(* Logix 5000 project; controller Lab5 vendor 1 type 14 code 54 rev 16.20; software revision 16.03 *)

TASK MainTask (continuous, watchdog 500 ms) : MainProgram

MODULES
   Local : vendor 1 type 14 code 54 (ICP 0, rev 16.20)
       : vendor 1 type 7 code 2 (ICP 5, rev 3.1, Input RPI 20 ms)
       : 1756-OB16D (ICP 6, rev 3.1, Output RPI 20 ms)
END_MODULES

PROGRAM MainProgram   (* main routine MainRoutine *)
VAR
   Forward_Start_Pushbutton : ALIAS FOR Local:5:I.Data.0;
   M1_Forward_Motor_Starter : ALIAS FOR Local:6:O.Data.0;
   M2_Reverse_Motor_Starter : ALIAS FOR Local:6:O.Data.1;
   Motor_Running_Light : ALIAS FOR Local:6:O.Data.2;
   Motor_Stopped_Light : ALIAS FOR Local:6:O.Data.3;
   Reverse_Start_Pushbutton : ALIAS FOR Local:5:I.Data.1;
   srtbh : TIMER;
   Stop_Pushbutton : ALIAS FOR Local:5:I.Data.2;
   Time_Motor_Not_Running : TIMER;
   Time_Motor_Running : TIMER;
   Timer1 : TIMER := (PRE := 10000);
   Timer_Motor_Not_Running : TIMER := (PRE := 99999999, ACC := 3844);
   Timer_Motor_Running : TIMER := (PRE := 999999999);
   Toggle_Switch_1 : ALIAS FOR Local:5:I.Data.3;
   Toggle_Switch_2 : ALIAS FOR Local:5:I.Data.4;
END_VAR

ROUTINE MainRoutine   (* ladder *)
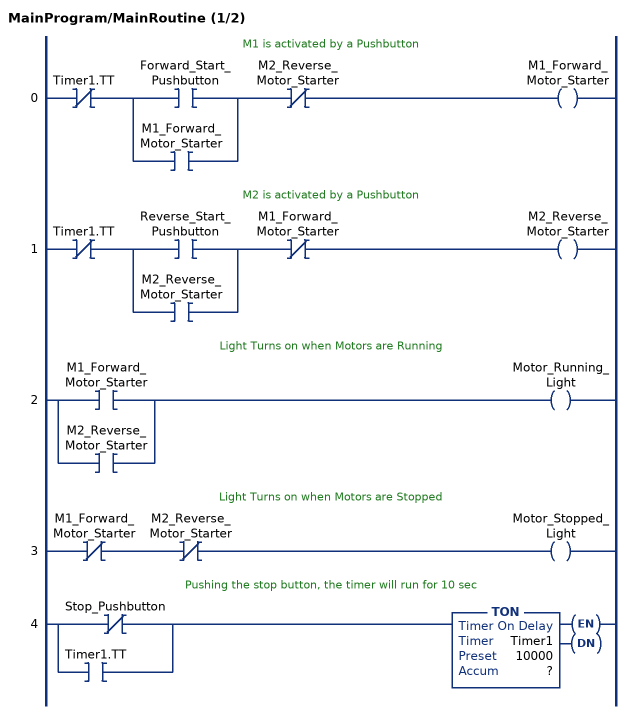
   // M1 is activated by a Pushbutton
   0: XIO(Timer1.TT)[XIC(Forward_Start_Pushbutton) ,XIC(M1_Forward_Motor_Starter) ]XIO(M2_Reverse_Motor_Starter)OTE(M1_Forward_Motor_Starter);
   // M2 is activated by a Pushbutton
   1: XIO(Timer1.TT)[XIC(Reverse_Start_Pushbutton) ,XIC(M2_Reverse_Motor_Starter) ]XIO(M1_Forward_Motor_Starter)OTE(M2_Reverse_Motor_Starter);
   // Light Turns on when Motors are Running
   2: [XIC(M1_Forward_Motor_Starter) ,XIC(M2_Reverse_Motor_Starter) ]OTE(Motor_Running_Light);
   // Light Turns on when Motors are Stopped
   3: XIO(M1_Forward_Motor_Starter)XIO(M2_Reverse_Motor_Starter)OTE(Motor_Stopped_Light);
   // Pushing the stop button, the timer will run for 10 sec
   4: [XIO(Stop_Pushbutton) ,XIC(Timer1.TT) ]TON(Timer1,?,?);
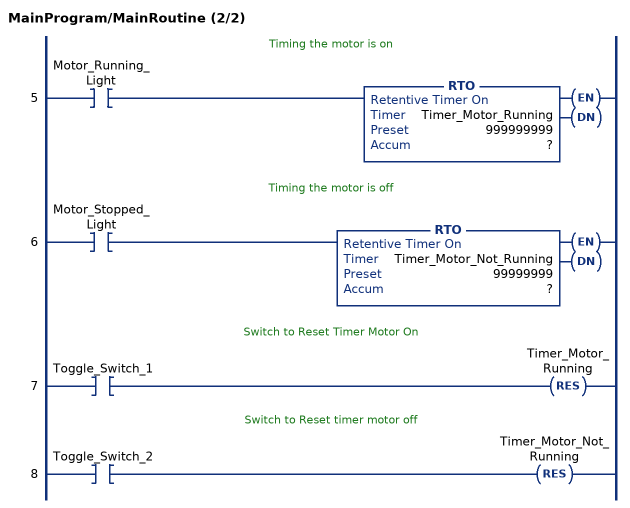
   // Timing the motor is on
   5: XIC(Motor_Running_Light)RTO(Timer_Motor_Running,?,?);
   // Timing the motor is off
   6: XIC(Motor_Stopped_Light)RTO(Timer_Motor_Not_Running,?,?);
   // Switch to Reset Timer Motor On
   7: XIC(Toggle_Switch_1)RES(Timer_Motor_Running);
   // Switch to Reset timer motor off
   8: XIC(Toggle_Switch_2)RES(Timer_Motor_Not_Running);
END_ROUTINE
END_PROGRAM
